Yaskawa INFORM job: LTRCKOF.JBI

/JOB
//NAME LTRCKOF
//POS
///NPOS 0,0,0,0,0,0
//INST
///DATE 2001/04/20 22:07
///ATTR SC,RW,MC
///GROUP1 RB1,BS1
///LVARS 1,0,0,0,0,0,0,0
NOP
'--- LT mode ----
GETARG LB000 IARG#(1)
JUMP *skip IF LB000<>1
SKILLSND "LSRCHOF"
SKILLSND "LTRACKOF"
ADVINIT
*skip
END
